// TIA Portal V19 export
DATA_BLOCK "Data_block_1"   // DB1
{ S7_Optimized_Access := 'TRUE' }
// stored: MemoryReserve 100
BEGIN
END_DATA_BLOCK
